// TwinCAT 3 PLC project RoboConnect_Tests_Runner
// ProgramVersion: 3.1.4024.0
// libraries:
//   Intecre.Utilities, * (Intecre Ltd)
//   mobject-collections, * (mobject)
//   RoboConnect, * (RoboConnect)
//   RoboConnect.Tests, * (RoboConnect)
//   Tc2_Standard, * (Beckhoff Automation GmbH)
//   Tc2_System, * (Beckhoff Automation GmbH)
//   Tc3_Module, * (Beckhoff Automation GmbH)
//   tcl_SimpleUnitTestLibrary, * (Red Rock Controls Limited)
// project tree:
//   CommandInvoker/ T_CommandInvoker_InvokesCommand_ProcessingTrue.TcPOU
//   CommandQueue/AddCommandToQueueQueueIncrementBy1/ T_CommandQueue_AddHighPriority_QueueIncrementedBy1.TcPOU, T_CommandQueue_AddNormalPriority_QueueIncrementedBy1.TcPOU, T_CommandQueue_AddLowPriority_QueueIncrementedBy1.TcPOU
//   CommandQueue/AddCommandToQueueReturnTrue/ T_CommandQueue_AddHighPriority_ReturnTrue.TcPOU, T_CommandQueue_AddLowPriority_ReturnTrue.TcPOU, T_CommandQueue_AddNormalPriority_ReturnTrue.TcPOU
//   CommandQueue/ClearCommandQueue/ T_CommandQueue_ClearWithHighPriority_ReturnTrue.TcPOU, T_CommandQueue_ClearWithNormalPriority_ReturnTrue.TcPOU, T_CommandQueue_ClearWithLowPriority_ReturnTrue.TcPOU, T_CommandQueue_ClearWithAllPriority_ReturnTrue.TcPOU
//   CommandQueue/GetNextCommand/ T_CommandQueue_GetNextCommandHighPriority_ReturnTrue.TcPOU, T_CommandQueue_GetNextCommandLowPriority_ReturnTrue.TcPOU, T_CommandQueue_GetNextCommandNormalPriority_ReturnTrue.TcPOU, T_CommandQueue_GetNextCommanHighPriorityWithNormalPriority_ReturnTrue.TcPOU, T_CommandQueue_GetNextCommandNormalPriorityWithLowPriority_ReturnTrue.TcPOU
//   CommandQueue/ T_MobjectQueue_AddItem_AddsItem.TcPOU
//   / GlobalTextList.TcGTLO, MAIN.TcPOU, PlcTask.TcTTO, T_MockCommandTask.TcPOU, Visualization Manager.TcVMO (not stored)
//   Task/ T_TaskBase_TaskDone_True.TcPOU, T_MockTask.TcPOU
//   TcpConnector/ T_TcpConnectTask_Connects.TcPOU, T_TcpConnectTask_Connects_1.TcPOU
//   VISUs/ TestUI.TcVIS
// (motion and I/O tree: see PLC project roboconnect)
// real-time tasks:
//   TASK PlcTask: cycle T#10ms, priority 22, ADS port 350
//   TASK PlcTask1: cycle T#10ms, priority 21, ADS port 351

CONFIGURATION RoboConnect_Tests_Runner
    RESOURCE PLC ON TwinCAT3
        TASK PlcTask(INTERVAL := T#10ms, PRIORITY := 21);
        PROGRAM MAIN WITH PlcTask : MAIN;
    END_RESOURCE
END_CONFIGURATION

// ---- MAIN.TcPOU
PROGRAM MAIN
VAR
  // Robot
  robot : T_MockRoboConnect;
  connectionTime : TIME := T#0.23S; // duration of simulated connection, for mock
  responseTime : TIME := T#0.8S;
  initialised : BOOL;

  testRunner : T_TestRunner;

  // Task Tests
  taskTestSuite : T_TestSuite;
  TaskBase_TaskDone_True : T_TaskBase_TaskDone_True(taskTestSuite);
  
  // CommandInvoker Tests
  commandInvokerTestSuite : T_testSuite;
  CommandInvoker_InvokesCommand_True : T_CommandInvoker_InvokesCommand_ProcessingTrue(commandInvokerTestSuite);
  
  // CommandQueueTests
  commandQueueTestSuite : T_TestSuite;

  CommandQueue_AddLowPriority_ReturnTrue : T_CommandQueue_AddLowPriority_ReturnTrue(commandQueueTestSuite);
  CommandQueue_AddNormalPriority_ReturnTrue : T_CommandQueue_AddNormalPriority_ReturnTrue(commandQueueTestSuite);
  CommandQueue_AddHighPriority_ReturnTrue : T_CommandQueue_AddHighPriority_ReturnTrue(commandQueueTestSuite);

  CommandQueue_AddHighPriority_QueueIncrementBy1 : T_CommandQueue_AddHighPriority_QueueIncrementedBy1(commandQueueTestSuite);
  CommandQueue_AddNormalPriority_QueueIncrementBy1 : T_CommandQueue_AddNormalPriority_QueueIncrementedBy1(commandQueueTestSuite);
  CommandQueue_AddLowPriority_QueueIncrementBy1 : T_CommandQueue_AddLowPriority_QueueIncrementedBy1(commandQueueTestSuite);

  CommandQueue_ClearWithHighPriority_ReturnTrue : T_CommandQueue_ClearWithHighPriority_ReturnTrue(commandQueueTestSuite);
  CommandQueue_ClearWithNormalPriority_ReturnTrue : T_CommandQueue_ClearWithNormalPriority_ReturnTrue(commandQueueTestSuite);
  CommandQueue_ClearWithLowPriority_ReturnTrue : T_CommandQueue_ClearWithLowPriority_ReturnTrue(commandQueueTestSuite);
  CommandQueue_ClearWithAllPriority_ReturnTrue : T_CommandQueue_ClearWithAllPriority_ReturnTrue(commandQueueTestSuite);

  CommandQueue_GetNextCommandHighPriority_ReturnTrue : T_CommandQueue_GetNextCommandHighPriority_ReturnTrue(commandQueueTestSuite);
  CommandQueue_GetNextCommandNormalPriority_ReturnTrue : T_CommandQueue_GetNextCommandNormalPriority_ReturnTrue(commandQueueTestSuite);
  CommandQueue_GetNextCommandLowPriority_ReturnTrue : T_CommandQueue_GetNextCommandLowPriority_ReturnTrue(commandQueueTestSuite);
  CommandQueue_GetNextCommanHighPriorityWithNormalPriority_ReturnTrue :T_CommandQueue_GetNextCommanHighPriorityWithNormalPriority_ReturnTrue(commandQueueTestSuite);
  CommandQueue_GetNextCommandNormalPriorityWithLowPriority_ReturnTrue :T_CommandQueue_GetNextCommandNormalPriorityWithLowPriority_ReturnTrue(commandQueueTestSuite);

  CommandQueue_MobjectQueue_AddItem_AddsItem : T_MobjectQueue_AddItem_AddsItem(commandQueueTestSuite);

  // RoboConnect Tests
  RoboConnectTestSuite : T_TestSuite;
  RoboConnect_WhenCalledWithLowTimeout_FailsConnection :
    T_RoboConnect_WhenCalledWithLowTimeout_FailsConnection(TestSuite := RoboConnectTestSuite, robot := robot, timeout := connectionTime - T#0.1S);
  RoboConnect_WhenCalled_IsConnectedTrue :
    T_RoboConnect_WhenCalled_IsConnectedTrue(TestSuite := RoboConnectTestSuite, robot := robot, timeout := connectionTime + T#0.1S);

  RoboConnect_SetAnalogOutput_IncorrectIndexFails : T_RoboConnect_SetAnalogOutput_IncorrectIndexFails(RoboConnectTestSuite, robot := robot, 999);
  RoboConnect_SetDigitalOutput_IncorrectIndexFails : T_RoboConnect_SetDigitalOutput_IncorrectIndexFails(RoboConnectTestSuite, robot := robot, 999);
  RoboConnect_SetToolAnalogOutput_IncorrectIndexFails : T_RoboConnect_SetToolAnalogOutput_IncorrectIndexFails(RoboConnectTestSuite, robot := robot, 999);
  RoboConnect_SetToolDigitalOutput_IncorrectIndexFails : T_RoboConnect_SetToolDigitalOutput_IncorrectIndexFails(RoboConnectTestSuite, robot := robot, 999);
  RoboConnect_GetAnalogOutput_IncorrectIndexFails : T_RoboConnect_GetAnalogOutput_IncorrectIndexFails(RoboConnectTestSuite, robot := robot, 999);
  RoboConnect_GetDigitalOutput_IncorrectIndexFails : T_RoboConnect_GetDigitalOutput_IncorrectIndexFails(RoboConnectTestSuite, robot := robot, 999);
  RoboConnect_GetToolAnalogOutput_IncorrectIndexFails : T_RoboConnect_GetToolAnalogOutput_IncorrectIndexFails(RoboConnectTestSuite, robot := robot, 999);
  RoboConnect_GetToolDigitalOutput_IncorrectIndexFails : T_RoboConnect_GetToolDigitalOutput_IncorrectIndexFails(RoboConnectTestSuite, robot := robot, 999);

  RoboConnect_SetAnalogOutput_CorrectIndexPasses : T_RoboConnect_SetAnalogOutput_CorrectIndexPasses(RoboConnectTestSuite, robot := robot, 1);
  RoboConnect_SetDigitalOutput_CorrectIndexPasses : T_RoboConnect_SetDigitalOutput_CorrectIndexPasses(RoboConnectTestSuite, robot := robot, 1);
  RoboConnect_SetToolAnalogOutput_CorrectIndexPasses : T_RoboConnect_SetToolAnalogOutput_CorrectIndexPasses(RoboConnectTestSuite, robot := robot, 1);
  RoboConnect_SetToolDigitalOutput_CorrectIndexPasses : T_RoboConnect_SetToolDigitalOutput_CorrectIndexPasses(RoboConnectTestSuite, robot := robot, 1);
  RoboConnect_GetAnalogOutput_CorrectIndexPasses : T_RoboConnect_GetAnalogOutput_CorrectIndexPasses(RoboConnectTestSuite, robot := robot, 1);
  RoboConnect_GetDigitalOutput_CorrectIndexPasses : T_RoboConnect_GetDigitalOutput_CorrectIndexPasses(RoboConnectTestSuite, robot := robot, 1);
  RoboConnect_GetToolAnalogOutput_CorrectIndexPasses : T_RoboConnect_GetToolAnalogOutput_CorrectIndexPasses(RoboConnectTestSuite, robot := robot, 1);
  RoboConnect_GetToolDigitalOutput_CorrectIndexPasses : T_RoboConnect_GetToolDigitalOutput_CorrectIndexPasses(RoboConnectTestSuite, robot := robot, 1);

  RoboConnect_GetDigitalOutput_ReturnsTrueOutput : T_RoboConnect_SetDigitalOutput_CorrectIndexPasses(RoboConnectTestSuite, robot, 1);
  RoboConnect_SetDigitalOutputTimeout_Fails : T_RoboConnect_SetDigitalOutputTimeout_Fails(RoboConnectTestSuite, robot, 1, T#1S);
  RoboConnect_GetToolDigitalOutput_ReturnsTrueOutput : T_RoboConnect_SetDigitalOutput_CorrectIndexPasses(RoboConnectTestSuite, robot, 1);
  RoboConnect_SetToolDigitalOutputTimeout_Fails : T_RoboConnect_SetDigitalOutputTimeout_Fails(RoboConnectTestSuite, robot, 1, T#1S);
  RoboConnect_GetAnalogOutput_ReturnsTrueOutput : T_RoboConnect_SetAnalogOutput_CorrectIndexPasses(RoboConnectTestSuite, robot, 1);
  RoboConnect_SetAnalogOutputTimeout_Fails : T_RoboConnect_SetToolAnalogOutput_TimeoutFails(RoboConnectTestSuite, robot, 1, T#1S);
  RoboConnect_GetToolAnalogOutput_ReturnsTrueOutput : T_RoboConnect_SetAnalogOutput_CorrectIndexPasses(RoboConnectTestSuite, robot, 1);
  RoboConnect_SetToolAnalogOutputTimeout_Fails : T_RoboConnect_SetToolAnalogOutput_TimeoutFails(RoboConnectTestSuite, robot, 1, T#1S);

END_VAR

IF NOT initialised THEN
  robot.SetConnectionTime(connectionTime);
  robot.SetGeneralCommandResponseDuration(responseTime);
  initialised := TRUE;
END_IF

IF testRunner.ReloadTests THEN
  testRunner.ClearTests();
  testRunner.AddTestSuite(taskTestSuite);
  testRunner.AddTestSuite(RoboConnectTestSuite);  
  testRunner.AddTestSuite(commandQueueTestSuite);
  testRunner.ReloadTests := FALSE;

END_IF

testRunner();
robot.CyclicLogic();

END_PROGRAM

// ---- Task/T_TaskBase_TaskDone_True.TcPOU
FUNCTION_BLOCK T_TaskBase_TaskDone_True EXTENDS T_UnitTestBase
VAR
  task : I_Task;
  myTestState, prevState : (INIT, ARRANGE, ACT, ASSERT) := INIT;
  taskRunner : T_MockTask;
  actual, expected : BOOL;
  counter : UINT;
END_VAR

taskRunner.CyclicLogic();

CASE myTestState OF
  INIT:
    StateChanged();
    myTestState := ARRANGE;

  ARRANGE:
    StateChanged();
    expected := TRUE;
    myTestState := ACT;
    
  ACT:
    IF StateChanged() THEN
      task := taskRunner.DoSomething(20);
    END_IF

    IF NOT WaitForCycles(30) THEN
      RETURN;
    END_IF

    myTestState := ASSERT;
    
  ASSERT:
    actual := task.Done;
    assertion.AssertEquals_BOOL(expected, actual, 'Task.Done = TRUE');
    myTestState := INIT;
    TestFinished();

END_CASE

METHOD PRIVATE StateChanged : BOOL
IF  myTestState = prevState THEN
  RETURN;
END_IF

prevState := myTestState;
StateChanged := TRUE;
END_METHOD

METHOD WaitForCycles : BOOL
VAR_INPUT
  maxCount : UINT;
END_VAR
counter := counter + 1;

IF counter = maxCount THEN
  counter := 0;
  WaitForCycles := TRUE;
END_IF
END_METHOD

END_FUNCTION_BLOCK

// ---- Task/T_MockTask.TcPOU
FUNCTION_BLOCK T_MockTask IMPLEMENTS I_Task
VAR_INPUT
  _busy : BOOL;
  _done : BOOL;
  _error : BOOL;
END_VAR
VAR
  state, prevState : (IDLE_STATE, BUSY_STATE, DONE_STATE, ERROR_STATE);
  counter : UINT := 0;
  cycleCount : UINT := 0;
END_VAR

METHOD Abort
// no op
END_METHOD

{warning 'add property implementation'}
PROPERTY Available : BOOL
GET
END_GET
END_PROPERTY

PROPERTY Busy : BOOL
GET
Busy := _busy;
END_GET
END_PROPERTY

METHOD PUBLIC CauseError
state := ERROR_STATE;
END_METHOD

METHOD PUBLIC CyclicLogic
CASE state OF
  IDLE_STATE:
    IF StateChanged() THEN
      _Busy := FALSE;
      _Done := FALSE;
      _Error := FALSE;
    END_IF
    
  BUSY_STATE:
    IF StateChanged() THEN
      _Busy := TRUE;
      _Done := FALSE;
      _Error := FALSE;
    END_IF

    IF NOT WaitForCycles(cycleCount) THEN
      RETURN;
    END_IF

    state := DONE_STATE;

  DONE_STATE:
    IF StateChanged() THEN
      _Busy := FALSE;
      _Done := TRUE;
      _Error := FALSE;
    END_IF

  ERROR_STATE:
    IF StateChanged() THEN
      _Error := TRUE;
      _Busy := FALSE;
      _Done := FALSE;
    END_IF

END_CASE
END_METHOD

PROPERTY Done : BOOL
GET
Done := _done;
END_GET
END_PROPERTY

METHOD PUBLIC DoSomething : I_Task
VAR_INPUT
  busyCycles : UINT;
END_VAR
state := BUSY_STATE;
cycleCount := busyCycles;
DoSomething := THIS^;
END_METHOD

PROPERTY Error : BOOL
GET
Error := _error;
END_GET
END_PROPERTY

{warning 'add property implementation'}
PROPERTY ErrorId : STRING
GET
END_GET
END_PROPERTY

METHOD Execute : BOOL
// no ops
END_METHOD

{warning 'add method implementation '}
METHOD Free
END_METHOD

METHOD PRIVATE StateChanged : BOOL
IF  state = prevState THEN
  RETURN;
END_IF

prevState := state;
StateChanged := TRUE;
END_METHOD

{warning 'add property implementation'}
PROPERTY Timeout : BOOL
GET
END_GET
END_PROPERTY

METHOD PRIVATE WaitForCycles : BOOL
VAR_INPUT
  maxCount : UINT;
END_VAR
counter := counter + 1;

IF counter = maxCount THEN
  counter := 0;
  WaitForCycles := TRUE;
END_IF
END_METHOD

END_FUNCTION_BLOCK

// ---- CommandInvoker/T_CommandInvoker_InvokesCommand_ProcessingTrue.TcPOU
FUNCTION_BLOCK T_CommandInvoker_InvokesCommand_ProcessingTrue EXTENDS T_UnitTestBase
VAR
  command : T_MockCommandTask;
  commandQueue : T_CommandQueue;
  commandInvoker : T_CommandInvoker;
  myTestState, prevState : (ARRANGE, ACT, ASSERT);
  actual : BOOL;
  expected : BOOL := TRUE;
END_VAR

CASE myTestState OF
  ARRANGE:
    myTestState := ACT;

  ACT:
    commandInvoker.Initialise(commandQueue);
    commandInvoker.CyclicLogic();
    command.initalise('test');
    commandQueue.AddNormalPriority(command);
    commandInvoker.CyclicLogic();
    myTestState := ASSERT;

  ASSERT:
    actual := commandInvoker.Processing;
    assertion.AssertEquals_UINT(expected, actual, 'actual := command.Busy;');
    myTestState := ARRANGE;
    TestFinished();
END_CASE

END_FUNCTION_BLOCK

// ---- T_MockCommandTask.TcPOU
FUNCTION_BLOCK  T_MockCommandTask EXTENDS T_NamedBase IMPLEMENTS I_CommandTask
VAR
	_busy : BOOL := FALSE;
	_error : BOOL := FALSE;
	_done : BOOL := FALSE;
  _timeout : BOOL := FALSE;
  _available : BOOL := TRUE;
  _errorId : STRING;
  _comPort : I_Connection;
  _msg : T_Maxstring;
  timeoutTimer : TON := (PT := TASK_TIMEOUT);
  
  state, prevState : (UNINITLIASED, INITALISED, EXECUTING, DONE_STATE, ERROR_STATE);
  
END_VAR
VAR CONSTANT 
  TASK_TIMEOUT : TIME := RoboConnectParams.TimeOut;
END_VAR

METHOD Abort
END_METHOD

PROPERTY Available : BOOL
GET
Available := _available;
END_GET
END_PROPERTY

PROPERTY Busy : BOOL
GET
Busy := _Busy;
END_GET
END_PROPERTY

METHOD PUBLIC CyclicLogic



CASE state OF
  UNINITLIASED:
    StateChanged();

  INITALISED:
    IF StateChanged() THEN
      logInfo('task initlaised');
    END_IF

  EXECUTING:
    IF StateChanged() THEN
      LogInfo('task executing');
      _busy := TRUE;
      timeoutTimer.IN := TRUE;
      
      IF NOT _comPort.Send(_msg) THEN
        state := ERROR_STATE;
        RETURN;
			END_IF
      
    END_IF
    
    IF timeoutTimer.Q THEN
      state := ERROR_STATE;
      LogError('Command timed out');
		END_IF

    IF _comPort.SendDone THEN
      state := DONE_STATE;
    END_IF

  DONE_STATE:
    IF StateChanged() THEN
      LogInfo('task done');
      _busy := FALSE;
      _done := TRUE;
      timeoutTimer.IN := FALSE;
    END_IF

  ERROR_STATE:
    IF StateChanged() THEN
      LogError('task error');
      _error := TRUE;
      _busy := FALSE;
      _done := FALSE;
    END_IF

END_CASE

timeoutTimer();
END_METHOD

PROPERTY Done : BOOL
GET
Done := _Done;
END_GET
END_PROPERTY

PROPERTY Error : BOOL
GET
Error := _Error;
END_GET
END_PROPERTY

PROPERTY PUBLIC ErrorId : string
GET
ErrorId := _errorId;
END_GET
END_PROPERTY

METHOD PUBLIC Execute : BOOL
IF state <> INITALISED THEN
  RETURN;
END_IF

state := EXECUTING;
EXECUTE := TRUE;
END_METHOD

METHOD PUBLIC Free
_Busy := FALSE;
_Error := FALSE;
_Done := FALSE;
 _timeout := FALSE;
 _available := TRUE;
  
_comPort := 0;
_msg := '';
END_METHOD

METHOD PUBLIC Initalise : BOOL
VAR_INPUT
 msg : T_Maxstring;
END_VAR
_done := FALSE;
_msg := msg;
state := INITALISED;
_available := FALSE;
Initalise := TRUE;
END_METHOD

METHOD PRIVATE StateChanged : BOOL
IF  state = prevState THEN
  RETURN;
END_IF

prevState := state;
StateChanged := TRUE;
END_METHOD

PROPERTY Timeout : BOOL
GET
Timeout := _timeout;
END_GET
END_PROPERTY

END_FUNCTION_BLOCK

// ---- CommandQueue/AddCommandToQueueReturnTrue/T_CommandQueue_AddLowPriority_ReturnTrue.TcPOU
FUNCTION_BLOCK T_CommandQueue_AddLowPriority_ReturnTrue EXTENDS T_UnitTestBase
VAR
  command : T_CommandTask;
  commandQueue : T_CommandQueue;
  myTestState, prevState : (ARRANGE, ACT, ASSERT);
  actual : BOOL := TRUE;
  expected : BOOL := TRUE;
END_VAR

CASE myTestState OF
  ARRANGE:
    myTestState := ACT;

  ACT:
    actual := commandQueue.AddLowPriority(command);
    myTestState := ASSERT;

  ASSERT:
    assertion.AssertEquals_BOOL(expected, actual, 'commandQueue.AddLowPriority = TRUE');
    myTestState := ARRANGE;
    TestFinished();
END_CASE

END_FUNCTION_BLOCK

// ---- CommandQueue/AddCommandToQueueReturnTrue/T_CommandQueue_AddNormalPriority_ReturnTrue.TcPOU
FUNCTION_BLOCK T_CommandQueue_AddNormalPriority_ReturnTrue EXTENDS T_UnitTestBase
VAR
  command : T_CommandTask;
  commandQueue : T_CommandQueue;
  myTestState, prevState : (ARRANGE, ACT, ASSERT);
  actual : BOOL := TRUE;
  expected : BOOL := TRUE;
END_VAR

CASE myTestState OF
  ARRANGE:
    myTestState := ACT;

  ACT:
    actual := commandQueue.AddNormalPriority(command);
    myTestState := ASSERT;

  ASSERT:
    assertion.AssertEquals_BOOL(expected, actual, 'commandQueue.AddNormalPriority = TRUE');
    myTestState := ARRANGE;
    TestFinished();
END_CASE

END_FUNCTION_BLOCK

// ---- CommandQueue/AddCommandToQueueReturnTrue/T_CommandQueue_AddHighPriority_ReturnTrue.TcPOU
FUNCTION_BLOCK T_CommandQueue_AddHighPriority_ReturnTrue EXTENDS T_UnitTestBase
VAR
  command : T_CommandTask;
  commandQueue : T_CommandQueue;
  myTestState, prevState : (ARRANGE, ACT, ASSERT);
  actual : BOOL := TRUE;
  expected : BOOL := TRUE;
END_VAR

CASE myTestState OF
  ARRANGE:
    myTestState := ACT;

  ACT:
    actual := commandQueue.AddHighPriority(command);
    myTestState := ASSERT;

  ASSERT:
    assertion.AssertEquals_BOOL(expected, actual, 'commandQueue.AddHighPriority = TRUE');
    myTestState := ARRANGE;
    TestFinished();
END_CASE

END_FUNCTION_BLOCK

// ---- CommandQueue/AddCommandToQueueQueueIncrementBy1/T_CommandQueue_AddHighPriority_QueueIncrementedBy1.TcPOU
FUNCTION_BLOCK T_CommandQueue_AddHighPriority_QueueIncrementedBy1 EXTENDS T_UnitTestBase
VAR
  command : T_MockCommandTask;
  commandQueue : T_CommandQueue;
  myTestState, prevState : (ARRANGE, ACT, ASSERT);
  actual : UINT;
  expected : UINT;
END_VAR

CASE myTestState OF
  ARRANGE:
  	expected := commandQueue.Count +1;
    myTestState := ACT;

  ACT:
    commandQueue.AddHighPriority(command);
	actual := commandQueue.Count;
    myTestState := ASSERT;

  ASSERT:
    assertion.AssertEquals_UINT(expected, actual, 'queue.count = queue.count +1');
    myTestState := ARRANGE;
    TestFinished();
END_CASE

END_FUNCTION_BLOCK

// ---- CommandQueue/AddCommandToQueueQueueIncrementBy1/T_CommandQueue_AddNormalPriority_QueueIncrementedBy1.TcPOU
FUNCTION_BLOCK T_CommandQueue_AddNormalPriority_QueueIncrementedBy1 EXTENDS T_UnitTestBase
VAR
  command : T_CommandTask;
  commandQueue : T_CommandQueue;
  myTestState, prevState : (ARRANGE, ACT, ASSERT);
  actual : UINT;
  expected : UINT;
END_VAR

CASE myTestState OF
  ARRANGE:
  	expected := commandQueue.Count +1;
    myTestState := ACT;

  ACT:
    commandQueue.AddNormalPriority(command);
	actual := commandQueue.Count;
    myTestState := ASSERT;

  ASSERT:
    assertion.AssertEquals_UINT(expected, actual, 'queue.count = queue.count +1');
    myTestState := ARRANGE;
    TestFinished();
END_CASE

END_FUNCTION_BLOCK

// ---- CommandQueue/AddCommandToQueueQueueIncrementBy1/T_CommandQueue_AddLowPriority_QueueIncrementedBy1.TcPOU
FUNCTION_BLOCK T_CommandQueue_AddLowPriority_QueueIncrementedBy1 EXTENDS T_UnitTestBase
VAR
  command : T_MockCommandTask;
  commandQueue : T_CommandQueue; //not sure if it needs to be .low.count
  myTestState, prevState : (ARRANGE, ACT, ASSERT);
  actual : UINT;
  expected : UINT;
END_VAR

CASE myTestState OF
  ARRANGE:
  	expected := commandQueue.Count +1;
    myTestState := ACT;

  ACT:
    commandQueue.AddLowPriority(command);
	actual := commandQueue.Count;
    myTestState := ASSERT;

  ASSERT:
    assertion.AssertEquals_UINT(expected, actual, 'queue.count = queue.count +1');
    myTestState := ARRANGE;
    TestFinished();
END_CASE

END_FUNCTION_BLOCK

// ---- CommandQueue/ClearCommandQueue/T_CommandQueue_ClearWithHighPriority_ReturnTrue.TcPOU
FUNCTION_BLOCK T_CommandQueue_ClearWithHighPriority_ReturnTrue EXTENDS T_UnitTestBase
VAR
  command : T_CommandTask;
  commandQueue : T_CommandQueue;
  myTestState, prevState : (ARRANGE, ACT, ASSERT);
  actual : UINT := 0;
  expected : UINT := 0;
END_VAR

CASE myTestState OF
  ARRANGE:
	commandQueue.AddHighPriority(command);
    myTestState := ACT;
  
  ACT:
    commandQueue.clear();
    actual := commandQueue.Count;
	myTestState := ASSERT;
	
  ASSERT:
  	
    assertion.AssertEquals_UINT(expected, actual, 'commandQueue.clear High Priority = TRUE');
    myTestState := ARRANGE;
    TestFinished();
END_CASE

END_FUNCTION_BLOCK

// ---- CommandQueue/ClearCommandQueue/T_CommandQueue_ClearWithNormalPriority_ReturnTrue.TcPOU
FUNCTION_BLOCK T_CommandQueue_ClearWithNormalPriority_ReturnTrue EXTENDS T_UnitTestBase
VAR
  command : T_CommandTask;
  commandQueue : T_CommandQueue;
  myTestState, prevState : (ARRANGE, ACT, ASSERT);
  actual : UINT := 0;
  expected : UINT := 0;
END_VAR

CASE myTestState OF
  ARRANGE:  
	commandQueue.AddNormalPriority(command);
  	myTestState := ACT;
	
  ACT:
    commandQueue.clear();
    actual := commandQueue.Count;
	myTestState := ASSERT;
	
  ASSERT:
    assertion.AssertEquals_UINT(expected, actual, 'commandQueue.clear Normal Priority = TRUE');
    myTestState := ARRANGE;
    TestFinished();
END_CASE

END_FUNCTION_BLOCK

// ---- CommandQueue/ClearCommandQueue/T_CommandQueue_ClearWithLowPriority_ReturnTrue.TcPOU
FUNCTION_BLOCK T_CommandQueue_ClearWithLowPriority_ReturnTrue EXTENDS T_UnitTestBase
VAR
  command : T_CommandTask;
  commandQueue : T_CommandQueue;
  myTestState, prevState : (ARRANGE, ACT, ASSERT);
  actual : UINT := 0;
  expected : UINT := 0;
END_VAR

CASE myTestState OF
  ARRANGE:
	commandQueue.AddLowPriority(command);
    myTestState := ACT;
  
  ACT:
    commandQueue.clear();
    actual := commandQueue.Count;
	myTestState := ASSERT;
	
  ASSERT:
    assertion.AssertEquals_UINT(expected, actual, 'commandQueue.clear Low Priority = TRUE');
    myTestState := ARRANGE;
    TestFinished();
END_CASE

END_FUNCTION_BLOCK

// ---- CommandQueue/ClearCommandQueue/T_CommandQueue_ClearWithAllPriority_ReturnTrue.TcPOU
FUNCTION_BLOCK T_CommandQueue_ClearWithAllPriority_ReturnTrue EXTENDS T_UnitTestBase
VAR
  commandLow : T_CommandTask;
  commandNormal : T_CommandTask;
  commandHigh : T_CommandTask;
  
  commandQueue : T_CommandQueue;
  myTestState, prevState : (ARRANGE, ACT, ASSERT);
  actual : UINT;
  expected : UINT;
END_VAR

CASE myTestState OF
  ARRANGE:
	commandQueue.AddHighPriority(commandHigh);
	commandQueue.AddNormalPriority(commandNormal);
  	commandQueue.AddLowPriority(commandLow);
	myTestState := ACT;
	
  ACT:
    commandQueue.clear();
	myTestState := ASSERT;
	
  ASSERT:
    assertion.AssertEquals_UINT(expected, actual, 'commandQueue.clear all Priority = TRUE');
    myTestState := ARRANGE;
    TestFinished();
END_CASE

END_FUNCTION_BLOCK

// ---- CommandQueue/GetNextCommand/T_CommandQueue_GetNextCommandHighPriority_ReturnTrue.TcPOU
FUNCTION_BLOCK T_CommandQueue_GetNextCommandHighPriority_ReturnTrue EXTENDS T_UnitTestBase
VAR
  command : T_CommandTask;
  commandQueue : T_CommandQueue;
  myTestState, prevState : (ARRANGE, ACT, ASSERT);
  actual : I_Task;
  expected : I_Task;
END_VAR

CASE myTestState OF
  ARRANGE:
  	expected := command;
	commandQueue.Clear();
	commandQueue.AddHighPriority(command);
    myTestState := ACT;
  
  ACT:
    commandQueue.GetNext(output_command => actual);
	myTestState := ASSERT;
	
  ASSERT:
    assertion.AssertEquals_INTERFACE(expected, actual, 'commandQueue.GetNext High priority = TRUE');
    myTestState := ARRANGE;
    TestFinished();
END_CASE

END_FUNCTION_BLOCK

// ---- CommandQueue/GetNextCommand/T_CommandQueue_GetNextCommandNormalPriority_ReturnTrue.TcPOU
FUNCTION_BLOCK T_CommandQueue_GetNextCommandNormalPriority_ReturnTrue EXTENDS T_UnitTestBase
VAR
  command :T_CommandTask;
  commandQueue : T_CommandQueue;
  myTestState, prevState : (ARRANGE, ACT, ASSERT);
  actual : I_Task;
  expected : I_Task;
END_VAR

CASE myTestState OF
  ARRANGE:
  	expected := command;
	commandQueue.Clear();
	commandQueue.AddNormalPriority(command);
    myTestState := ACT;
  
  ACT:
    commandQueue.GetNext(output_command => actual);
	myTestState := ASSERT;
	
  ASSERT:
    assertion.AssertEquals_INTERFACE(expected, actual, 'commandQueue.GetNext Normal priority = TRUE');
    myTestState := ARRANGE;
    TestFinished();
END_CASE

END_FUNCTION_BLOCK

// ---- CommandQueue/GetNextCommand/T_CommandQueue_GetNextCommandLowPriority_ReturnTrue.TcPOU
FUNCTION_BLOCK T_CommandQueue_GetNextCommandLowPriority_ReturnTrue EXTENDS T_UnitTestBase
VAR
  command : T_CommandTask;
  commandQueue : T_CommandQueue;
  myTestState, prevState : (ARRANGE, ACT, ASSERT);
  actual : I_Task;
  expected : I_Task;
END_VAR

CASE myTestState OF
  ARRANGE:
  	expected := command;
	commandQueue.Clear();
	commandQueue.AddLowPriority(command);
    myTestState := ACT;
  
  ACT:
    commandQueue.GetNext(output_command => actual);
	myTestState := ASSERT;
	
  ASSERT:
    assertion.AssertEquals_INTERFACE(expected, actual, 'commandQueue.GetNext Low priority = TRUE');
    myTestState := ARRANGE;
    TestFinished();
END_CASE

END_FUNCTION_BLOCK

// ---- CommandQueue/GetNextCommand/T_CommandQueue_GetNextCommanHighPriorityWithNormalPriority_ReturnTrue.TcPOU
FUNCTION_BLOCK T_CommandQueue_GetNextCommanHighPriorityWithNormalPriority_ReturnTrue EXTENDS T_UnitTestBase
VAR
  commandHighPriority : T_CommandTask;
  commandNormalPriority : T_CommandTask;
  commandQueue : T_CommandQueue;
  myTestState, prevState : (ARRANGE, ACT, ASSERT);
  actual : I_Task;
  expected : I_Task;
END_VAR

CASE myTestState OF
  ARRANGE:
  	expected := commandHighPriority;
	commandQueue.Clear();
	commandQueue.AddNormalPriority(commandNormalPriority);
	commandQueue.AddHighPriority(commandHighPriority);
    myTestState := ACT;
  
  ACT:
    commandQueue.GetNext(output_command => actual);
	myTestState := ASSERT;
	
  ASSERT:
    assertion.AssertEquals_INTERFACE(expected, actual, 'commandQueue.GetNext high priority with Low priority = TRUE');
    myTestState := ARRANGE;
    TestFinished();
END_CASE

END_FUNCTION_BLOCK

// ---- CommandQueue/GetNextCommand/T_CommandQueue_GetNextCommandNormalPriorityWithLowPriority_ReturnTrue.TcPOU
FUNCTION_BLOCK T_CommandQueue_GetNextCommandNormalPriorityWithLowPriority_ReturnTrue EXTENDS T_UnitTestBase
VAR
  commandLowPriority : T_CommandTask;
  commandNormalPriority : T_CommandTask;
  commandQueue : T_CommandQueue;
  myTestState, prevState : (ARRANGE, ACT, ASSERT);
  actual : I_Task;
  expected : I_Task;
END_VAR

CASE myTestState OF
  ARRANGE:
  	expected := commandNormalPriority;
	commandQueue.Clear();
	commandQueue.AddNormalPriority(commandNormalPriority);
	commandQueue.AddLowPriority(commandLowPriority);
    myTestState := ACT;
  
  ACT:
    commandQueue.GetNext(output_command => actual);
	myTestState := ASSERT;
	
  ASSERT:
    assertion.AssertEquals_INTERFACE(expected, actual, 'commandQueue.GetNext high priority with Low priority = TRUE');
    myTestState := ARRANGE;
    TestFinished();
END_CASE

END_FUNCTION_BLOCK

// ---- CommandQueue/T_MobjectQueue_AddItem_AddsItem.TcPOU
FUNCTION_BLOCK T_MobjectQueue_AddItem_AddsItem EXTENDS T_UnitTestBase
VAR_INPUT
END_VAR
VAR_OUTPUT
END_VAR
VAR
	Queue : Queue;
	queueLength : DINT;
	item : INT := 1;
END_VAR

Queue.AddItem(item);
queueLength := Queue.Count;
TestFinished();

END_FUNCTION_BLOCK

// ---- TcpConnector/T_TcpConnectTask_Connects.TcPOU
FUNCTION_BLOCK T_TcpConnectTask_Connects EXTENDS T_UnitTestBase
VAR
  ip : T_IPv4Addr;
  port : UINT;
  tcpipConnection : T_ConnectionTCPIP;
  
  myTestState, prevState : (ARRANGE, ACT, ASSERT);
  actual, expected : I_Task;
END_VAR

CASE myTestState OF
  ARRANGE:
    ip := '127.0.0.1';
    port := 5000;

  ACT:
    tcpipConnection.Connect();
    
    IF resultTask.Done THEN
      state := ARRANGE;
		END_IF

  ASSERT:
    actual := resultTask.Done;
    assertion.AssertEquals_BOOL(expected, actual, 'Task.Done = TRUE');
    myTestState := ARRANGE;
    TestFinished();

END_CASE

END_FUNCTION_BLOCK

// ---- TcpConnector/T_TcpConnectTask_Connects_1.TcPOU
FUNCTION_BLOCK T_TcpConnectTask_Connects_1 EXTENDS T_UnitTestBase
VAR
  ip : T_IPv4Addr;
  port : UINT;
  connectTask : T_SocketConnectTask;
  resultTask : I_Task;
  myTestState, prevState : (ARRANGE, ACT, ASSERT);
  
  actual, expected : BOOL;
END_VAR

CASE myTestState OF
  ARRANGE:
    ip := '127.0.0.1';
    port := 5000;

  ACT:
    connectTask.Execute(ip, port);
    
    // Cycles
    connectTask.CyclicLogic();
    connectTask.CyclicLogic();
    connectTask.CyclicLogic();
    
    IF resultTask.Done THEN
      state := ARRANGE;
		END_IF

  ASSERT:
    actual := resultTask.Done;
    assertion.AssertEquals_BOOL(expected, actual, 'Task.Done = TRUE');
    myTestState := ARRANGE;
    TestFinished();

END_CASE

END_FUNCTION_BLOCK

// ---- VISUs/TestUI.TcVIS
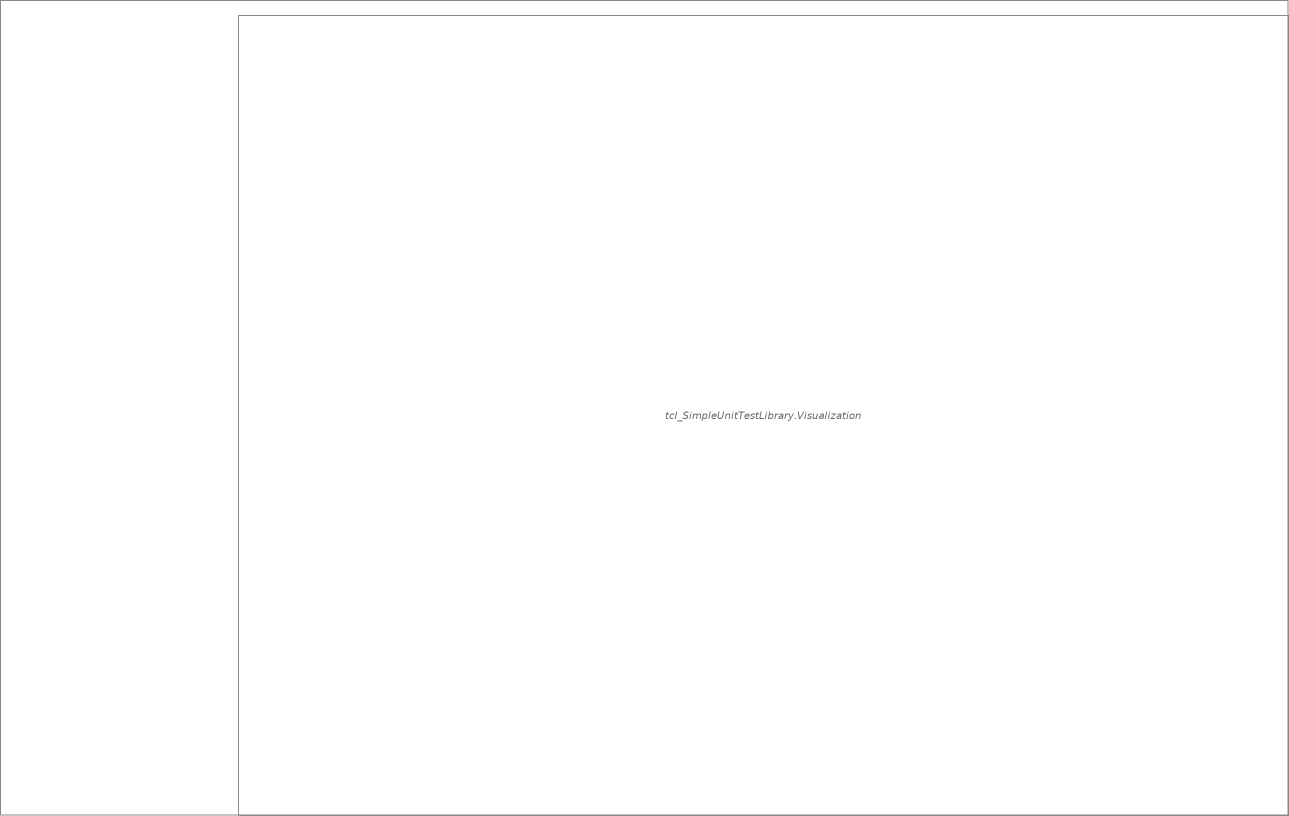
VISUALIZATION TestUI  // 1289x816
    Frame (238,15 1051x801)
        shows tcl_SimpleUnitTestLibrary.Visualization(TestRunner := MAIN.testRunner)
END_VISUALIZATION
